FUNCTION_BLOCK BasicControlTS5
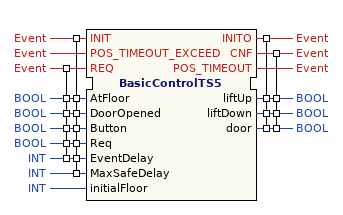
  EVENT_INPUT
    INIT WITH AtFloor, DoorOpened, Button, Req, EventDelay, MaxSafeDelay;
    POS_TIMEOUT_EXCEED;
    REQ WITH AtFloor, DoorOpened, Button, Req, EventDelay;
  END_EVENT
  EVENT_OUTPUT
    INITO WITH liftUp, liftDown, door;
    CNF WITH liftUp, liftDown, door;
    POS_TIMEOUT;
  END_EVENT
  VAR_INPUT
    AtFloor : BOOL;
    DoorOpened : BOOL;
    Button : BOOL;
    Req : BOOL;
    EventDelay : INT;
    MaxSafeDelay : INT;
    initialFloor : INT := 2;
  END_VAR
  VAR_OUTPUT
    liftUp : BOOL;
    liftDown : BOOL;
    door : BOOL;
  END_VAR
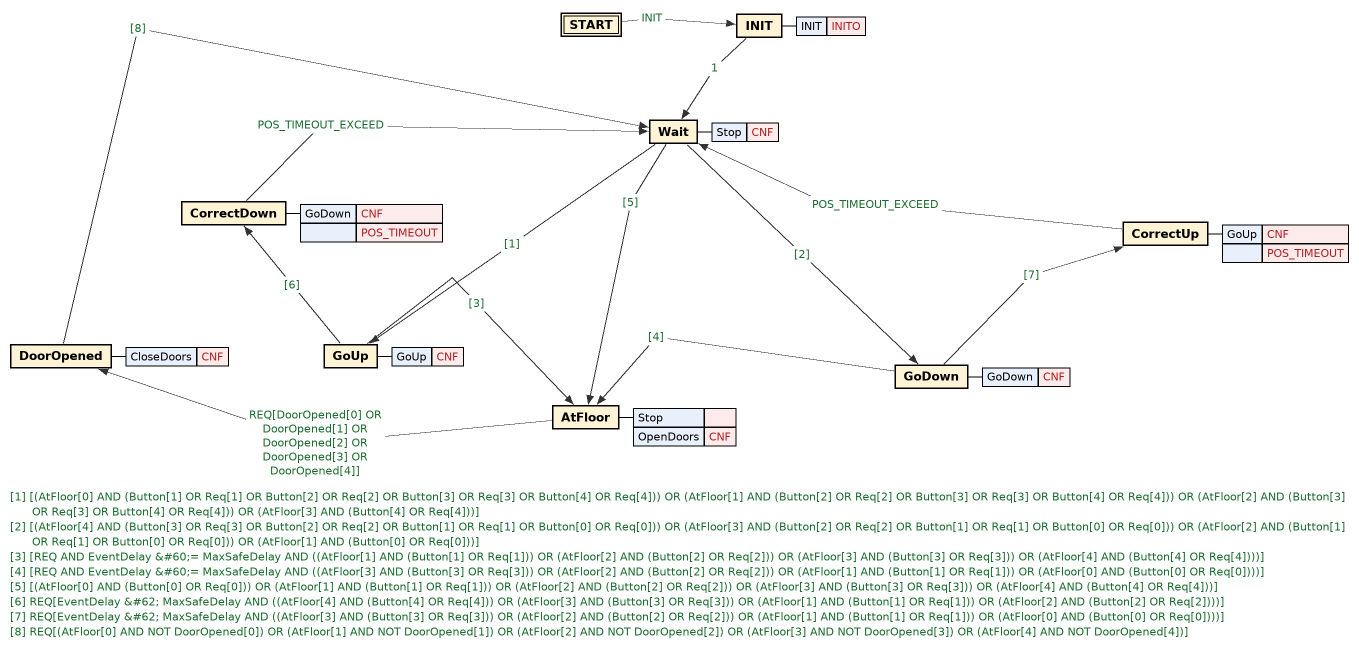
  EC_STATES
    START;
    INIT : INIT -> INITO;
    AtFloor : Stop, OpenDoors -> CNF;
    GoUp : GoUp -> CNF;
    Wait : Stop -> CNF;
    DoorOpened : CloseDoors -> CNF;
    GoDown : GoDown -> CNF;
    CorrectDown : GoDown -> CNF, -> POS_TIMEOUT;
    CorrectUp : GoUp -> CNF, -> POS_TIMEOUT;
  END_STATES
  EC_TRANSITIONS
    START TO INIT := INIT;
    INIT TO Wait := 1;
    GoUp TO AtFloor := [REQ AND EventDelay &#60;= MaxSafeDelay AND ((AtFloor[1] AND (Button[1] OR Req[1])) OR (AtFloor[2] AND (Button[2] OR Req[2])) OR (AtFloor[3] AND (Button[3] OR Req[3])) OR (AtFloor[4] AND (Button[4] OR Req[4])))];
    Wait TO AtFloor := [(AtFloor[0] AND (Button[0] OR Req[0])) OR (AtFloor[1] AND (Button[1] OR Req[1])) OR (AtFloor[2] AND (Button[2] OR Req[2])) OR (AtFloor[3] AND (Button[3] OR Req[3])) OR (AtFloor[4] AND (Button[4] OR Req[4]))];
    Wait TO GoUp := [(AtFloor[0] AND (Button[1] OR Req[1] OR Button[2] OR Req[2] OR Button[3] OR Req[3] OR Button[4] OR Req[4])) OR (AtFloor[1] AND (Button[2] OR Req[2] OR Button[3] OR Req[3] OR Button[4] OR Req[4])) OR (AtFloor[2] AND (Button[3] OR Req[3] OR Button[4] OR Req[4])) OR (AtFloor[3] AND (Button[4] OR Req[4]))];
    AtFloor TO DoorOpened := REQ[DoorOpened[0] OR DoorOpened[1] OR DoorOpened[2] OR DoorOpened[3] OR DoorOpened[4]];
    GoDown TO AtFloor := [REQ AND EventDelay &#60;= MaxSafeDelay AND ((AtFloor[3] AND (Button[3] OR Req[3])) OR (AtFloor[2] AND (Button[2] OR Req[2])) OR (AtFloor[1] AND (Button[1] OR Req[1])) OR (AtFloor[0] AND (Button[0] OR Req[0])))];
    GoUp TO CorrectDown := REQ[EventDelay &#62; MaxSafeDelay AND ((AtFloor[4] AND (Button[4] OR Req[4])) OR (AtFloor[3] AND (Button[3] OR Req[3])) OR (AtFloor[1] AND (Button[1] OR Req[1])) OR (AtFloor[2] AND (Button[2] OR Req[2])))];
    GoDown TO CorrectUp := REQ[EventDelay &#62; MaxSafeDelay AND ((AtFloor[3] AND (Button[3] OR Req[3])) OR (AtFloor[2] AND (Button[2] OR Req[2])) OR (AtFloor[1] AND (Button[1] OR Req[1])) OR (AtFloor[0] AND (Button[0] OR Req[0])))];
    Wait TO GoDown := [(AtFloor[4] AND (Button[3] OR Req[3] OR Button[2] OR Req[2] OR Button[1] OR Req[1] OR Button[0] OR Req[0])) OR (AtFloor[3] AND (Button[2] OR Req[2] OR Button[1] OR Req[1] OR Button[0] OR Req[0])) OR (AtFloor[2] AND (Button[1] OR Req[1] OR Button[0] OR Req[0])) OR (AtFloor[1] AND (Button[0] OR Req[0]))];
    DoorOpened TO Wait := REQ[(AtFloor[0] AND NOT DoorOpened[0]) OR (AtFloor[1] AND NOT DoorOpened[1]) OR (AtFloor[2] AND NOT DoorOpened[2]) OR (AtFloor[3] AND NOT DoorOpened[3]) OR (AtFloor[4] AND NOT DoorOpened[4])];
    CorrectUp TO Wait := POS_TIMEOUT_EXCEED;
    CorrectDown TO Wait := POS_TIMEOUT_EXCEED;
  END_TRANSITIONS
  ALGORITHM INIT IN ST:
liftDown := FALSE;&#38;#10;liftUp := FALSE;&#38;#10;
  END_ALGORITHM
  ALGORITHM GoDown IN ST:
liftDown := TRUE;&#38;#10;liftUp := FALSE;&#38;#10;
  END_ALGORITHM
  ALGORITHM Stop IN ST:
liftDown := FALSE;&#38;#10;liftUp := FALSE;&#38;#10;
  END_ALGORITHM
  ALGORITHM GoUp IN ST:
liftUp := TRUE;&#38;#10;liftDown := FALSE;&#38;#10;
  END_ALGORITHM
  ALGORITHM OpenDoors IN ST:
door[0] := AtFloor[0];&#38;#10;door[1] := AtFloor[1];&#38;#10;door[2] := AtFloor[2];&#38;#10;door[3] := AtFloor[3];&#38;#10;door[4] := AtFloor[4];&#38;#10;
  END_ALGORITHM
  ALGORITHM CloseDoors IN ST:
door[0] := FALSE;&#38;#10;door[1] := FALSE;&#38;#10;door[2] := FALSE;&#38;#10;door[3] := FALSE;&#38;#10;door[4] := FALSE;&#38;#10;
  END_ALGORITHM
END_FUNCTION_BLOCK
